// SIMATIC S7-200 project (STEP 7-Micro/WIN), CPU 221 REL 01.10

SYMBOL_TABLE USER1
den_1            Q0.0
den_2            Q0.1
den_3            Q0.2
den_4            Q0.3
den_5            Q0.4
den_6            Q0.5
den_7            Q0.6
den_8            Q0.7
den_9            Q1.0
den_10           Q1.1
bien             M0.0
END_SYMBOL_TABLE

ORGANIZATION_BLOCK MAIN:OB1
TITLE=PROGRAM COMMENTS
BEGIN
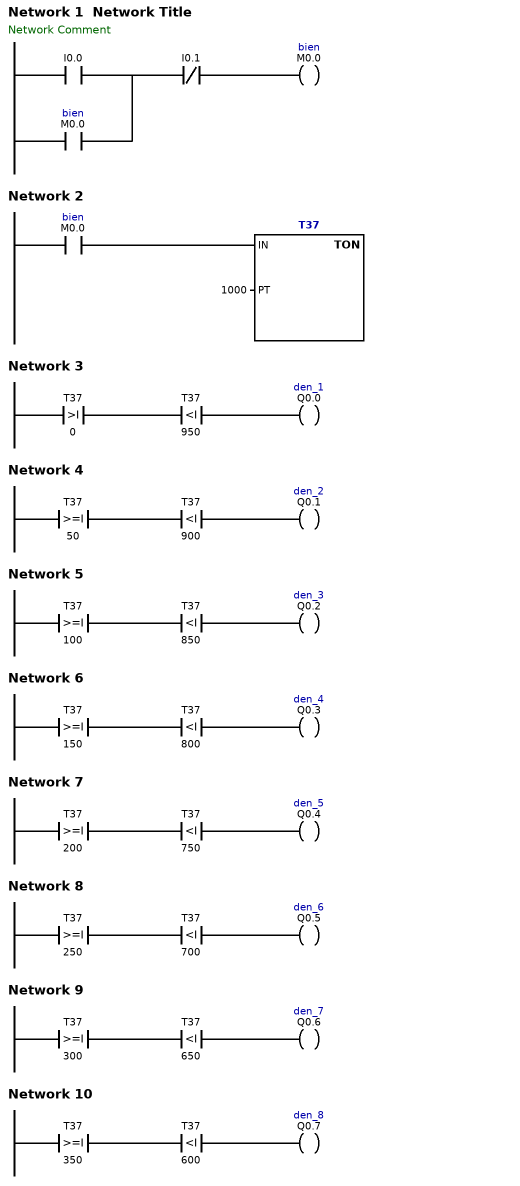
Network 1 // Network Title
// Network Comment
LD     I0.0
O      bien:M0.0
AN     I0.1
=      bien:M0.0
Network 2
LD     bien:M0.0
TON    T37, 1000
Network 3
LDW>   T37, 0
AW<    T37, 950
=      den_1:Q0.0
Network 4
LDW>=  T37, 50
AW<    T37, 900
=      den_2:Q0.1
Network 5
LDW>=  T37, 100
AW<    T37, 850
=      den_3:Q0.2
Network 6
LDW>=  T37, 150
AW<    T37, 800
=      den_4:Q0.3
Network 7
LDW>=  T37, 200
AW<    T37, 750
=      den_5:Q0.4
Network 8
LDW>=  T37, 250
AW<    T37, 700
=      den_6:Q0.5
Network 9
LDW>=  T37, 300
AW<    T37, 650
=      den_7:Q0.6
Network 10
LDW>=  T37, 350
AW<    T37, 600
=      den_8:Q0.7
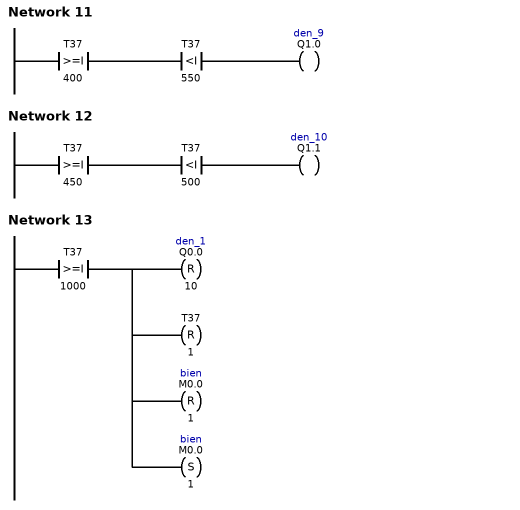
Network 11
LDW>=  T37, 400
AW<    T37, 550
=      den_9:Q1.0
Network 12
LDW>=  T37, 450
AW<    T37, 500
=      den_10:Q1.1
Network 13
LDW>=  T37, 1000
R      den_1:Q0.0, 10
R      T37, 1
R      bien:M0.0, 1
S      bien:M0.0, 1
END_ORGANIZATION_BLOCK
